FUNCTION_BLOCK FB_SetupRobot
VAR_INPUT
END_VAR
VAR_OUTPUT
END_VAR
VAR
	// setup arms, responsible for arm kinematic and control
	m_setupArms :ARRAY[1..g_sArmNum] OF FB_SetupArm;
	
	// arm state
	m_setupArmState:ARRAY[1..g_sArmNum] OF E_setupArmState:=[4(E_setupArmState.SetupArmState_Init)];
	m_lastSetupArmState:ARRAY[1..g_sArmNum] OF E_setupArmState:=[4(E_setupArmState.SetupArmState_Init)];
	m_nextSetupArmState:ARRAY[1..g_sArmNum] OF E_setupArmState:=[4(E_setupArmState.SetupArmState_Init)];
	
	// all arm controller instance 
	m_armCtrlFactory :ARRAY[1..g_sArmNum,1..SetupArmState_totalNum] OF I_SetupArmCtrl;
	m_armInit :ARRAY[1..g_sArmNum] OF FB_SetupCtrlInit;
	m_armError :ARRAY[1..g_sArmNum] OF FB_SetupCtrlError;
	m_armSelfCheck :ARRAY[1..g_sArmNum] OF FB_SetupCtrlSelfCheck;
	m_armHold :ARRAY[1..g_sArmNum] OF FB_SetupCtrlHold;
	m_armManualAdjust :ARRAY[1..g_sArmNum] OF FB_SetupCtrlManualAdjust;
	m_armAutoAdjust :ARRAY[1..g_sArmNum] OF FB_SetupCtrlAutoAdjust;
	m_armPackage :ARRAY[1..g_sArmNum] OF FB_SetupCtrlPackage;
	m_armCart :ARRAY[1..g_sArmNum] OF FB_SetupCtrlCart;
	m_armGraCali :ARRAY[1..g_sArmNum] OF FB_SetupCtrlGraCali;
	
	
	// arm controller interface
	m_armCtrl :ARRAY[1..g_sArmNum] OF I_SetupArmCtrl;
	m_armCtrlCmds :ARRAY[1..g_sArmNum] OF ST_SetupArmCtrlCmds;

END_VAR

METHOD PUBLIC getStatus : BOOL
VAR_IN_OUT
	// slave robot information, including arm status and cartesian data
	r_setupStatus :ST_SetupStatus;
	
	// slave robot joint data
	r_setupJointsData :ST_SetupJointData;
	
END_VAR

VAR
	i:INT;
END_VAR
r_setupStatus.m_armState:=m_setupArmState;

// TODO: project cartesion data to monitor coordinate
FOR i:=1 TO g_sArmNum DO
	
	// cartesion
	r_setupStatus.m_curEndPose[i]:=m_setupArms[i].curCartPose;
	r_setupStatus.m_rcPos[i]:=m_setupArms[i].rcPos;
	
	// joint
	r_setupJointsData.m_curMotorPos[i]:=m_setupArms[i].curMotorPos;
	r_setupJointsData.m_curLinkPos[i]:=m_setupArms[i].curLinkPos;
	r_setupJointsData.m_curJntPos[i]:=m_setupArms[i].curJntPos;
	r_setupJointsData.m_curJntVel[i]:=m_setupArms[i].curJntVel;
	r_setupJointsData.m_curJntTrq[i]:=m_setupArms[i].curJntTrq;
	
	// command info
	// joint info
	r_setupJointsData.m_cmdJntPos[i]:=m_armCtrlCmds[i].m_cmdJntPos;
	r_setupJointsData.m_cmdJntVel[i]:=m_armCtrlCmds[i].m_cmdJntVel;
	r_setupJointsData.m_cmdJntTrq[i]:=m_armCtrlCmds[i].m_cmdJntTrq;
	
END_FOR
END_METHOD

METHOD PUBLIC Init : BOOL
VAR_INPUT
END_VAR
VAR
	i:INT;
END_VAR
FOR i:=1 TO g_sArmNum DO
	// arm init
	m_setupArms[i].Init(i);
	m_setupArmState[i]:=SlaveArmState_Init;
	m_lastSetupArmState[i]:=SlaveArmState_Init;
	m_nextSetupArmState[i]:=SlaveArmState_Init;
	
	// command init
	m_armCtrlCmds[i].m_jntEnableFlag := g_zeroVec5i;
	m_armCtrlCmds[i].m_jntOPMode := g_setupAllPosMode;
	m_armCtrlCmds[i].m_cmdJntPos := m_setupArms[i].curJntPos;
	m_armCtrlCmds[i].m_cmdJntVel := g_zeroVec5d;
	m_armCtrlCmds[i].m_cmdJntAcc := g_zeroVec5d;
	m_armCtrlCmds[i].m_cmdJntTrq := g_zeroVec5d;
	
	// generate controller factory
	m_armCtrlFactory[i,SetupArmState_Error] := m_armError[i];
	m_armCtrlFactory[i,SetupArmState_Init] := m_armInit[i];
	m_armCtrlFactory[i,SetupArmState_SelfCheck] := m_armSelfCheck[i];
	m_armCtrlFactory[i,SetupArmState_Hold] := m_armHold[i];
	m_armCtrlFactory[i,SetupArmState_ManulAdjust] := m_armManualAdjust[i];
	m_armCtrlFactory[i,SetupArmState_AutoAdjust] := m_armAutoAdjust[i];
	m_armCtrlFactory[i,SetupArmState_Package] := m_armPackage[i];
	m_armCtrlFactory[i,SetupArmState_Cart] := m_armCart[i];
	m_armCtrlFactory[i,SetupArmState_GravityCali] := m_armGraCali[i];
	
	// assign controller
	m_armCtrl[i]:=m_armCtrlFactory[i,m_setupArmState[i]];
	m_armCtrl[i].Init(m_setupArms[i],m_armCtrlCmds[i]);
END_FOR
END_METHOD

METHOD PUBLIC run : BOOL
VAR_IN_OUT CONSTANT
	i_setupInputDataPool:ST_SetupInputDataPool;
END_VAR
VAR
	i:INT;
END_VAR
// state machine transition
stateMachine(i_setupInputDataPool);

FOR i:=1 TO g_sArmNum DO
	// update dynamic data
	m_setupArms[i].updateDyna(i_setupInputDataPool.m_setupJnt3Gravity, i_setupInputDataPool.m_setupJnt5Gravity);
								
	// update slave arm kinematics
	m_setupArms[i].updateStatus();
	
	// null ptr check
	IF 0 = m_armCtrl[i] THEN
		EXIT;
	END_IF
	
	// run controller
	m_armCtrl[i].run(m_setupArms[i],m_armCtrlCmds[i]);

	// update commands to drivers
	m_setupArms[i].updateCmds(m_armCtrlCmds[i]);

END_FOR
END_METHOD

// state machine check and transit 
METHOD PROTECTED stateMachine : BOOL
VAR_IN_OUT CONSTANT
		i_setupInputDataPool:ST_SetupInputDataPool;
END_VAR
VAR
	i:INT;
END_VAR
FOR i:=1 TO g_sArmNum DO
	// State machine transit 
	CASE m_setupArmState[i] OF
		// init
		SetupArmState_Init:
			IF m_armCtrl[i].isFinished  THEN
				m_nextSetupArmState[i]:=SetupArmState_SelfCheck;
			END_IF

		//self check
		SetupArmState_SelfCheck:
			IF m_armCtrl[i].isFinished  THEN
				m_nextSetupArmState[i]:=SetupArmState_Hold;
			END_IF
		
		//hold
		SetupArmState_Hold:
			IF m_setupArms[i].manualAdjustOn THEN
				m_nextSetupArmState[i]:=SetupArmState_ManulAdjust;
			ELSIF m_setupArms[i].autoAdjustDir<>0 THEN
				m_nextSetupArmState[i]:=SetupArmState_AutoAdjust;
			END_IF
			
(*		
		//package
		SetupArmState_Package:
		
		//cart
		SetupArmState_Cart:
		
		//gravity calibration
		SetupArmState_GravityCali:
		
*)
	END_CASE
	
	// Controller transit
	IF m_nextSetupArmState[i]<> m_setupArmState[i] THEN
		// reset current controller
		m_armCtrl[i].reset();
		
		// transit to new controller
		m_lastSetupArmState[i]:=m_setupArmState[i];
		m_setupArmState[i]:=m_nextSetupArmState[i];
		m_armCtrl[i]:=m_armCtrlFactory[i,m_setupArmState[i]];
		
		// init next controller
		m_armCtrl[i].Init(m_setupArms[i],m_armCtrlCmds[i]);
		m_setupArms[i].updateCmds(m_armCtrlCmds[i]);
	END_IF
END_FOR
END_METHOD

END_FUNCTION_BLOCK

(* stored: Version 1.1.0.1, ProductVersion 3.1.4024.12
   POU FB_SetupRobot: Id {41d3f45b-28bf-4672-9f4d-c2ea05b7f776}, SpecialFunc None
   Method getStatus: Id {87cb863f-d525-453d-a0db-af97bcb1e34e}
   Method Init: Id {0db3a443-112b-48f7-898b-6b92ed428f2d}
   Method run: Id {00eef043-1869-4f40-8399-c0641788ce23}
   Method stateMachine: Id {ec1b7cf8-3c23-4752-ad51-56e56c84a99b} *)
